// TwinCAT 3 PLC project TcoIoBeckhoff
// Title: TcoIoBeckhoff
// Company: Vortex.Library
// ProjectVersion: 1.19.1.1780
// ProgramVersion: 3.1.4024.12
// libraries:
//   Tc2_Standard, * (Beckhoff Automation GmbH)
//   Tc2_System, * (Beckhoff Automation GmbH)
//   Tc3_Module, * (Beckhoff Automation GmbH)
// project tree:
//   Abstractions/AI/ AI_1_Module.TcPOU, AI_ChannelStatus.TcPOU (not stored), AI_Channel.TcPOU (not stored)
//   Abstractions/ InfoData.TcPOU (not stored), WcState.TcPOU (not stored)
//   GVLs/ IO.TcGVL
//   Modules/EL922x/FBs/ FuseChannelBasic.TcPOU, FuseChannelExtended.TcPOU, FuseModuleEL922x.TcPOU
//   Modules/EL922x/ITFs/ IFuseChannelBasic.TcIO, IFuseChannelExtended.TcIO (not stored)
//   Modules/EL922x/STs/ EL922x_ChannelBasic.TcDUT (not stored), EL922x_ChannelExtended.TcDUT (not stored), OutputStruct.TcDUT (not stored), StatusStructBasic.TcDUT, StatusStructExtended.TcDUT
//   / PlcTask.TcTTO
//   Version/ Global_Version.TcGVL (not stored)
// real-time tasks:
//   TASK PlcTask: cycle T#10ms, priority 20, ADS port 350
// I/O:
//   DEVICE Device 1 (EtherCAT) (disabled), AmsNetId 172.20.10.104.2.1
//     Term 1 (EK1100) [EK1100 EtherCAT Coupler (2A E-Bus)]
//       Term 2 (EL3001) [EL3001 1Ch. Ana. Input +/-10V]
//       Term 3 (EL9221-4030) [EL9221-4030 Overcurrent protection 24V DC, 1Ch., 3A]

CONFIGURATION TcoIoBeckhoff
    RESOURCE PLC ON TwinCAT3
        TASK PlcTask(INTERVAL := T#10ms, PRIORITY := 20);
        PROGRAM MAIN WITH PlcTask : MAIN;
    END_RESOURCE
END_CONFIGURATION

// ---- Modules/EL922x/STs/StatusStructBasic.TcDUT
TYPE StatusStructBasic :
STRUCT
		Enabled: BIT;
		Tripped : BIT;
		{attribute 'hide'}
		_hidden_bit_0: BIT;
		{attribute 'hide'}
		_hidden_bit_1: BIT;
		HWProtection : BIT;
		{attribute 'hide'}
		_hidden_bit_2: BIT;
		{attribute 'hide'}
		_hidden_bit_3: BIT;
		CurrentLevelWarning : BIT;
		
		CoolDownLock : BIT;
		{attribute 'hide'}
		_hidden_bit_4: BIT;
		{attribute 'hide'}
		_hidden_bit_5: BIT;
		{attribute 'hide'}
		_hidden_bit_6: BIT;
		Diag : BIT;
		TxPDOState : BIT;
		{attribute 'hide'}
		_hidden_bit_7: BIT;
		{attribute 'hide'}
		_hidden_bit_8: BIT;
		
		{attribute 'hide'}
		_hidden_bit_9: BIT;
		{attribute 'hide'}
		_hidden_bit_10: BIT;
		Error : BIT;
		StateReset : BIT;
		StateSwitch : BIT;
		{attribute 'hide'}
		_hidden_bit_11: BIT;
		{attribute 'hide'}
		_hidden_bit_12: BIT;
		{attribute 'hide'}
		_hidden_bit_13: BIT;
		{attribute 'hide'}
		_hidden_byte_14: BYTE;
END_STRUCT
END_TYPE

// ---- Modules/EL922x/STs/StatusStructExtended.TcDUT
TYPE StatusStructExtended :
STRUCT
	Enabled: BIT;
	Tripped : BIT;
	ShortCircuit : BIT;
	Overload : BIT;
	HWProtection : BIT;
	Overvoltage : BIT;
	Undervoltage : BIT;
	CurrentLevelWarning : BIT;
	
	CoolDownLock : BIT;
	DisabledBySwitch : BIT;
	DisabledByDI : BIT;
	DisabledByOutput : BIT;
	Diag : BIT;
	TxPDOState : BIT;
	InputCycleCount : BIT;
	InputCycleCount2 : BIT;
	
	StateDeviceSwitch : BIT;
	StateDigitalInput : BIT;
	Error : BIT;
	StateReset : BIT;
	StateSwitch : BIT;
	{attribute 'hide'}
	_hidden_bit_0: BIT;
	{attribute 'hide'}
	_hidden_bit_1: BIT;
	{attribute 'hide'}
	_hidden_bit_2: BIT;
	{attribute 'hide'}
	_hidden_byte_0: BYTE;
END_STRUCT
END_TYPE

// ---- GVLs/IO.TcGVL
{attribute 'qualified_only'}
VAR_GLOBAL 

_CX2040 : TcoHardwareDiagContext;

_EK1100 : EK1100;

//	{attribute 'iopath:"Device 1 (EtherCAT)\\Term 1 (EK1100)\\Term 2 (EL3001)"'}
//	_EL3001 : AI_1_Module;
	
	
//	_channel_1 : FuseChannelBasic;
//	_channel_2 : FuseChannelBasic;
	
//	{attribute 'iopath:"Device 1 (EtherCAT)\\Term 1 (EK1100)\\Term 3 (EL9221-4030)"'}
//	_EL922x : FuseModuleEL922x(_channel_1, _channel_2);

////	{attribute addProperty Name "A1"}
////	A1 	: EL6002;
	{attribute addProperty Name "A2"}
	A2 	: EL1809;
//	{attribute addProperty Name "A3"}
//	A3 	: EL2809;
////	{attribute addProperty Name "A4"}
////	A4 	: EL4004;
//	{attribute addProperty Name "A5"}
//	A5 	: EL2809;
////	{attribute addProperty Name "A6"}
////	A6 	: EL6001;

//2DI
_EL1002 : EL1002;
_EL1012 : EL1012;
_EL1052 : EL1052;
_EL1202 : EL1202;
_EL1252 : EL1252;
_EL1382 : EL1382;
_EL1502 : EL1502;
_EL1512 : EL1512;
_EL1702 : EL1702;
_EL1712 : EL1712;
_EL1722 : EL1722;
//4DI
_EL1004 : EL1004;
_EL1014 : EL1014;
_EL1024 : EL1024;
_EL1034 : EL1034;
_EL1054 : EL1054;
_EL1084 : EL1084;
_EL1094 : EL1094;
_EL1104 : EL1104;
_EL1114 : EL1114;
_EL1124 : EL1124;
_EL1134 : EL1134;
_EL1144 : EL1144;
_EL1254 : EL1254;
_EL1804 : EL1804;
_EL1814 : EL1814;
//8DI
_EL1008 : EL1008;
_EL1018 : EL1018;
_EL1088 : EL1088;
_EL1098 : EL1098;
_EL1808 : EL1808;
//16DI
_EL1809 : EL1809;
_EL1819 : EL1819;
_EL1852 : EL1852;
_EL1859 : EL1859;
_EL1862 : EL1862;
_EL1872 : EL1872;
_EL1889 : EL1889;
_EL1899 : EL1899;
//2DO
_EL2002 : EL2002;
_EL2022 : EL2022;
_EL2032 : EL2032;
_EL2042 : EL2042;
_EL2202 : EL2202;
_EL2252 : EL2252;
_EL2502 : EL2502;
_EL2521 : EL2521;
_EL2522 : EL2522;
_EL2535 : EL2535;
_EL2595 : EL2595;
_EL2596 : EL2596;
_EL2602 : EL2602;
_EL2612 : EL2612;
_EL2622 : EL2622;
_EL2652 : EL2652;
_EL2712 : EL2712;
_EL2722 : EL2722;
_EL2732 : EL2732;
//4DO
_EL2004 : EL2004;
_EL2014 : EL2014;
_EL2024 : EL2024;
_EL2034 : EL2034;
_EL2044 : EL2044;
_EL2084 : EL2084;
_EL2124 : EL2124;
_EL2624 : EL2624;
_EL2634 : EL2634;
_EL2784 : EL2784;
_EL2794 : EL2794;
//8DO
_EL2008 : EL2008;
_EL2088 : EL2088;
_EL2258 : EL2258;
_EL2788 : EL2788;
_EL2798 : EL2798;
_EL2808 : EL2808;
_EL2828 : EL2828;
_EL2878 : EL2878;
//16DO
_EL2809 : EL2809;
_EL2819 : EL2819;
_EL2872 : EL2872;
_EL2889 : EL2889;

//1AI
_EL3001 : EL3001;
_EL3011 : EL3011;
_EL3021 : EL3021;
_EL3041 : EL3041;
_EL3051 : EL3051;
_EL3061 : EL3061;
_EL3101 : EL3101;
_EL3111 : EL3111;
_EL3121 : EL3121;
_EL3141 : EL3141;
_EL3151 : EL3151;
_EL3161 : EL3161;
_EL3201 : EL3201;
_EL3311 : EL3311;
_EL3351 : EL3351;
_EL3356 : EL3356;
_EL3681 : EL3681;

//2AI
_EL3002 : EL3002;
_EL3012 : EL3012;
_EL3022 : EL3022;
_EL3042 : EL3042;
_EL3052 : EL3052;
_EL3062 : EL3062;
_EL3102 : EL3102;
_EL3112 : EL3112;
_EL3122 : EL3122;
_EL3142 : EL3142;
_EL3152 : EL3152;
_EL3162 : EL3162;
_EL3182 : EL3182;
_EL3202 : EL3202;
_EL3312 : EL3312;
_EL3602 : EL3602;
_EL3612 : EL3612;
_EL3692 : EL3692;

//3AI
_EL3403 : EL3403;
_EL3413 : EL3413;
_EL3423 : EL3423;
_EL3433 : EL3433;
_EL3443 : EL3443;
_EL3453 : EL3453;
_EL3483 : EL3483;

//4AI
_EL3004 : EL3004;
_EL3014 : EL3014;
_EL3024 : EL3024;
_EL3044 : EL3044;
_EL3054 : EL3054;
_EL3064 : EL3064;
_EL3104 : EL3104;
_EL3114 : EL3114;
_EL3124 : EL3124;
_EL3144 : EL3144;
_EL3154 : EL3154;
_EL3164 : EL3164;
_EL3174 : EL3174;
_EL3204 : EL3204;
_EL3214 : EL3214;
_EL3314 : EL3314;

//5AI
_EL3255 : EL3255;

//6AI
_EL3446 : EL3446;

//8AI
_EL3008 : EL3008;
_EL3048 : EL3048;
_EL3058 : EL3058;
_EL3068 : EL3068;
_EL3208 : EL3208;
_EL3218 : EL3218;
_EL3318 : EL3318;

//1AO
_EL4001 : EL4001;
_EL4011 : EL4011;
_EL4021 : EL4021;
_EL4031 : EL4031;

//2AO
_EL4002 : EL4002;
_EL4012 : EL4012;
_EL4022 : EL4022;
_EL4032 : EL4032;
_EL4102 : EL4102;
_EL4112 : EL4112;
_EL4122 : EL4122;
_EL4132 : EL4132;

//4AO
_EL4004 : EL4004;
_EL4014 : EL4014;
_EL4024 : EL4024;
_EL4034 : EL4034;
_EL4104 : EL4104;
_EL4114 : EL4114;
_EL4124 : EL4124;
_EL4134 : EL4134;

//8AO
_EL4008 : EL4008;
_EL4018 : EL4018;
_EL4028 : EL4028;
_EL4038 : EL4038;

//EL5xx1
_EL5001 : EL5001;
_EL5021 : EL5021;
_EL5101 : EL5101;
_EL5151 : EL5151;

//EL5xx2
_EL5002 : EL5002;
_EL5032 : EL5032;
_EL5042 : EL5042;
_EL5072 : EL5072;
_EL5102 : EL5102;
_EL5112 : EL5112;
_EL5122 : EL5122;
_EL5152 : EL5152;

//EL6xx1
_EL6001 : EL6001;
_EL6002 : EL6002;
_EL6021 : EL6021;
_EL6022 : EL6022;
_EL6070 : EL6070;
_EL6601 : EL6601;
_EL6614 : EL6614;
_EL6631 : EL6631;
_EL6731 : EL6731;
_EL6751 : EL6751;


END_VAR

// ---- Modules/EL922x/ITFs/IFuseChannelBasic.TcIO
INTERFACE IFuseChannelBasic EXTENDS __SYSTEM.IQueryInterface

PROPERTY CoolDownLock  : bool
GET
END_GET
END_PROPERTY

PROPERTY CurrentLevelWarning  : bool
GET
END_GET
END_PROPERTY

PROPERTY Diag  : bool
GET
END_GET
END_PROPERTY

PROPERTY Enabled : bool
GET
END_GET
END_PROPERTY

PROPERTY Error  : bool
GET
END_GET
END_PROPERTY

PROPERTY HardwareProtection : bool
GET
END_GET
END_PROPERTY

METHOD ResetFuse : BOOL
END_METHOD

PROPERTY StateReset : bool
GET
END_GET
END_PROPERTY

PROPERTY StateSwitch : bool
GET
END_GET
END_PROPERTY

METHOD SwitchFuse : BOOL
END_METHOD

PROPERTY Tripped : bool
GET
END_GET
END_PROPERTY

PROPERTY TxPDOState  : bool
GET
END_GET
END_PROPERTY

END_INTERFACE

// ---- Abstractions/AI/AI_1_Module.TcPOU
FUNCTION_BLOCK AI_1_Module
VAR
	{attribute addProperty Name  "1"}
	iCHANNEL_1 : AI_Channel;
	{attribute addProperty Name  "WcState"}
	WcState : WcState;
	{attribute addProperty Name  "WcState"}
	InfoData : WcState;
END_VAR

END_FUNCTION_BLOCK

// ---- Modules/EL922x/FBs/FuseChannelBasic.TcPOU
FUNCTION_BLOCK FuseChannelBasic IMPLEMENTS IFuseChannelBasic
VAR_INPUT
END_VAR
VAR_OUTPUT
END_VAR
VAR
	_Chn : EL922x_ChannelBasic;	
END_VAR


PROPERTY CoolDownLock : BOOL
GET
CoolDownLock := _Chn.Status.CoolDownLock;
END_GET
END_PROPERTY


PROPERTY CurrentLevelWarning : BOOL
GET
CurrentLevelWarning := _Chn.Status.CurrentLevelWarning;
END_GET
END_PROPERTY


PROPERTY Diag : BOOL
GET
Diag := _Chn.Status.Diag;
END_GET
END_PROPERTY


PROPERTY Enabled : BOOL
GET
Enabled := _Chn.Status.Enabled;
END_GET
END_PROPERTY


PROPERTY Error : BOOL
GET
Error := _Chn.Status.Error;
END_GET
END_PROPERTY


PROPERTY HardwareProtection : BOOL
GET
HardwareProtection := _Chn.Status.HWProtection;
END_GET
END_PROPERTY


METHOD ResetFuse : BOOL
_Chn.Control.Reset := NOT _Chn.Control.Reset;
END_METHOD


PROPERTY StateReset : BOOL
GET
StateReset := _Chn.Status.StateReset;
END_GET
END_PROPERTY


PROPERTY StateSwitch : BOOL
GET
StateSwitch := _Chn.Status.StateSwitch;
END_GET
END_PROPERTY

METHOD SwitchFuse : BOOL
_Chn.Control.Switch := NOT _Chn.Control.Switch;
END_METHOD


PROPERTY Tripped : BOOL
GET
Tripped := _Chn.Status.Tripped;
END_GET
END_PROPERTY


PROPERTY TxPDOState : BOOL
GET
TxPDOState := _Chn.Status.TxPDOState;
END_GET
END_PROPERTY

END_FUNCTION_BLOCK

// ---- Modules/EL922x/FBs/FuseModuleEL922x.TcPOU
FUNCTION_BLOCK FuseModuleEL922x
VAR_INPUT
END_VAR
VAR_OUTPUT
END_VAR
VAR
	_chn1Basic : IFuseChannelBasic;
	_chn2Basic : IFuseChannelBasic;
	_chn1Extended : IFuseChannelExtended;
	_chn2Extended : IFuseChannelExtended;	
END_VAR

METHOD FB_init : BOOL
VAR_INPUT
	bInitRetains : BOOL; // if TRUE, the retain variables are initialized (warm start / cold start)
	bInCopyCode : BOOL;  // if TRUE, the instance afterwards gets moved into the copy code (online change)
	chn1 : IFuseChannelBasic;
	chn2 : IFuseChannelBasic;
END_VAR
_chn1Basic := chn1;
__QUERYINTERFACE(_chn1Basic, _chn1Extended);
_chn2Basic := chn2;
__QUERYINTERFACE(_chn2Basic, _chn2Extended);
END_METHOD

END_FUNCTION_BLOCK

// ---- Modules/EL922x/FBs/FuseChannelExtended.TcPOU
FUNCTION_BLOCK FuseChannelExtended EXTENDS FuseChannelBasic IMPLEMENTS IFuseChannelExtended
VAR_INPUT
END_VAR
VAR_OUTPUT
END_VAR
VAR
	_ChnEx : EL922x_ChannelExtended;	
END_VAR


PROPERTY DisabledByDI : BOOL
GET
DisabledByDI := _ChnEx.Status.DisabledByDI;
END_GET
END_PROPERTY


PROPERTY DisabledByOutput : BOOL
GET
DisabledByOutput := _ChnEx.Status.DisabledByOutput;
END_GET
END_PROPERTY


PROPERTY DisabledBySwitch : BOOL
GET
DisabledBySwitch := _ChnEx.Status.DisabledBySwitch;
END_GET
END_PROPERTY


PROPERTY Overload : BOOL
GET
Overload := _ChnEx.Status.Overload;
END_GET
END_PROPERTY


PROPERTY Overvoltage : BOOL
GET
Overvoltage := _ChnEx.Status.Overvoltage;
END_GET
END_PROPERTY

{warning 'add property implementation'}
PROPERTY ShortCircuit : BOOL
GET
ShortCircuit := _ChnEx.Status.ShortCircuit;
END_GET
END_PROPERTY

{warning 'add property implementation'}
PROPERTY StateDeviceSwitch : BOOL
GET
StateDeviceSwitch := _ChnEx.Status.StateDeviceSwitch;
END_GET
END_PROPERTY

{warning 'add property implementation'}
PROPERTY StateDigitalInput : BOOL
GET
StateDigitalInput := _ChnEx.Status.StateDigitalInput;
END_GET
END_PROPERTY

{warning 'add property implementation'}
PROPERTY Undervoltage : BOOL
GET
Undervoltage := _ChnEx.Status.Undervoltage;
END_GET
END_PROPERTY

END_FUNCTION_BLOCK
